SYSTEM test
  (* Version 1.0, 2026-08-26, Grafinger *)
  APPLICATION testApp
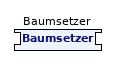
    SUBAPPS
      Baumsetzer : FBs::Baumsetzer::Baumsetzer;
    END_SUBAPPS
  END_APPLICATION
  DEVICE FORTE_PC : iec61499::system::FORTE_PC(MGR_ID := "192.168.4.1:61499" (* Device manager socket ID *))
    {SET_ATTRIBUTE(Profile, HOLOBLOC)}
    RESOURCE EMB_RES : iec61499::system::EMB_RES
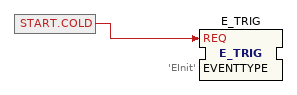
      FBS
        E_TRIG : iec61499::events::E_TRIG(EVENTTYPE := 'EInit');
      END_FBS
      EVENT_CONNECTIONS
        START.COLD TO E_TRIG.REQ;
      END_CONNECTIONS
    END_RESOURCE
  END_DEVICE
  MAPPINGS
    testApp.Baumsetzer ON FORTE_PC.EMB_RES;
  END_MAPPINGS
  SEGMENTS
    Ethernet : iec61499::system::Ethernet;
  END_SEGMENTS
  LINKS
    FORTE_PC => Ethernet;
  END_LINKS
END_SYSTEM
